(* IEC 61131-3 sources: BuildVersion/BuildVer, 5 files *)

(* ---- DT_TO_ISO.st ---- *)
(* TODO: Add your comment here *)
FUNCTION DT_TO_ISO

	Str	:=	'';

	DT_TO_DTStructure(DT1,ADR(DT1Struct));
	sVar	:=	UINT_TO_STRING(DT1Struct.year);
	Str	:=	CONCAT(Str,sVar);
	Str	:=	CONCAT(Str,'-');

	sVar	:=	USINT_TO_STRING(DT1Struct.month);
	IF DT1Struct.month < 10 THEN
		Str	:=	CONCAT(Str,'0');
	END_IF;
	Str	:=	CONCAT(Str,sVar);
	Str	:=	CONCAT(Str,'-');

	sVar	:=	USINT_TO_STRING(DT1Struct.day);
	IF DT1Struct.day < 10 THEN
		Str	:=	CONCAT(Str,'0');
	END_IF;
	Str	:=	CONCAT(Str,sVar);
	Str	:=	CONCAT(Str,'T');

	sVar	:=	USINT_TO_STRING(DT1Struct.hour);
	IF DT1Struct.hour < 10 THEN
		Str	:=	CONCAT(Str,'0');
	END_IF;
	Str	:=	CONCAT(Str,sVar);
	Str	:=	CONCAT(Str,':');

	sVar	:=	USINT_TO_STRING(DT1Struct.minute);
	IF DT1Struct.minute < 10 THEN
		Str	:=	CONCAT(Str,'0');
	END_IF;
	Str	:=	CONCAT(Str,sVar);
	Str	:=	CONCAT(Str,':');

	sVar	:=	USINT_TO_STRING(DT1Struct.second);
	IF DT1Struct.second < 10 THEN
		Str	:=	CONCAT(Str,'0');
	END_IF;
	Str	:=	CONCAT(Str,sVar);
	Str	:=	CONCAT(Str,'.000Z');

	brsmemcpy(pStr,ADR(Str),length);
	DT_TO_ISO	:=	LEN(Str);

END_FUNCTION

(* ---- actLogVersion.st ---- *)
ACTION actLogVersion:

	GetLogbookIdent.Name := '$$arlogusr';
	GetLogbookIdent.Execute := TRUE;
	GetLogbookIdent();

	Message := BuildVersion.Git.Describe;
	Message := CONCAT(Message, ' (');
	Message := CONCAT(Message, BuildVersion.Git.Branch);
	Message := CONCAT(Message, ', ');

	IF BuildVersion.Git.ChangeWarning THEN
		WriteToLogbook.EventID := ArEventLogMakeEventID(arEVENTLOG_SEVERITY_WARNING, 400, 10000);
		//WriteToLogbook.EventID := ArEventLogMakeEventID(arEVENTLOG_SEVERITY_WARNING, 0, 0);
		Message := CONCAT(Message, 'dirty, ');
	ELSE
		WriteToLogbook.EventID := ArEventLogMakeEventID(arEVENTLOG_SEVERITY_INFO, 400, 10000);
		//WriteToLogbook.EventID := ArEventLogMakeEventID(arEVENTLOG_SEVERITY_INFO, 0, 0);
		Message := CONCAT(Message, 'clean, ');
	END_IF;

	DT_TO_ISO(BuildVersion.Project.BuildDateUTC,ADR(sBuildDate),SIZEOF(sBuildDate));
	Message := CONCAT(Message, sBuildDate);
	Message := CONCAT(Message, ')');

	WriteToLogbook.AddDataSize := LEN(Message) + 1;

	WriteToLogbook.Ident := GetLogbookIdent.Ident;
	WriteToLogbook.AddDataFormat := arEVENTLOG_ADDFORMAT_TEXT;
	WriteToLogbook.AddData := ADR(Message);
	WriteToLogbook.ObjectID := 'BuildVersion';
	WriteToLogbook.Execute := TRUE;
	WriteToLogbook();

	GetLogbookIdent.Execute := FALSE;
	GetLogbookIdent();
	WriteToLogbook.Execute := FALSE;
	WriteToLogbook();

END_ACTION

(* ---- BuildVer.st ---- *)
(*********************************************************************************
 * Copyright: B&R Industrial Automation GmbH
 * Author:    pawlikb
 * Created:   April 10, 2026/8:08 AM
 * Based on original work by Tyler Matijevich
 *********************************************************************************)

PROGRAM _INIT

	//Always log during boot
	actLogVersion;

	//On update set alarm
	IF _Revision <> BuildVersion.Git.Describe OR _BuildDate <> BuildVersion.Project.BuildDate THEN
		_Revision	:=	BuildVersion.Git.Describe;
		_BuildDate	:=	BuildVersion.Project.BuildDate;
		//MpAlarmXSet(gAlarmXCore,'UpdateInstalled');
	END_IF;

END_PROGRAM

PROGRAM _CYCLIC

	//Bind to alarm
	BuildVersion.Git.ChangeWarning;

	//On update set alarm and log
	IF _Revision <> BuildVersion.Git.Describe OR _BuildDate <> BuildVersion.Project.BuildDate THEN
		_Revision	:=	BuildVersion.Git.Describe;
		_BuildDate	:=	BuildVersion.Project.BuildDate;
		//MpAlarmXSet(gAlarmXCore,'UpdateInstalled');

		actLogVersion;
	END_IF;

END_PROGRAM

(* ---- BuildVer.var ---- *)
VAR
	GetLogbookIdent : ArEventLogGetIdent;
	WriteToLogbook : ArEventLogWrite;
	Message : STRING[121];
END_VAR
VAR RETAIN
	_Revision : STRING[80];
	_BuildDate : DATE_AND_TIME;
END_VAR
VAR
	sBuildDate : STRING[80];
END_VAR

(* ---- LocalFunctions.fun ---- *)
{REDUND_ERROR} FUNCTION DT_TO_ISO : UDINT (*TODO: Add your comment here*) (*$GROUP=User,$CAT=User,$GROUPICON=User.png,$CATICON=User.png*)
	VAR_INPUT
		DT1 : DATE_AND_TIME;
		pStr : UDINT;
		length : UDINT;
	END_VAR
	VAR
		DT1Struct : DTStructure;
		sVar : STRING[25];
		Str : STRING[25];
	END_VAR
END_FUNCTION
